// Mitsubishi GX Works2 project: Project1   PLC: Q03UDV

PROGRAM MAIN
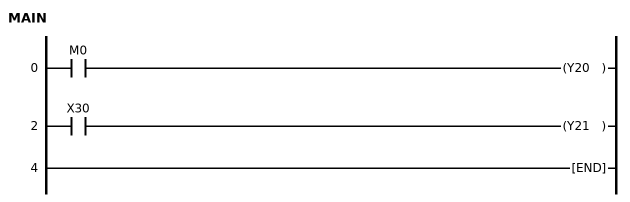
0     LD      M0
      OUT     Y20
2     LD      X30
      OUT     Y21
4     END
END_PROGRAM
